Fanuc KAREL source: ks00052.KL

-- PROVISIONAL review KL for V770-1; original PC SHA256 1c92deb38e2fccdaf37a37c3a64e49adf54957a86a3390e17938cd36c78a080f
-- Incomplete behavior may be omitted. Consult companion uncertainty JSON. Do not deploy.
PROGRAM KS00052
%NOLOCKGROUP
BEGIN
  -- UNRESOLVED_PC offsets 5-13; opcodes 3F,75
  -- UNRESOLVED_PC offsets 18-27; opcodes 3F,75
  -- UNRESOLVED_PC offsets 32-46; opcodes 22,22,1E
  -- UNRESOLVED_PC offsets 51-55; opcodes 7F
END KS00052
